// TIA Portal V16 export
// export: Created 2022-11-17T15:49:23.5959361Z, ExportSetting WithDefaults, DisplayName Totally Integrated Automation Portal, DisplayVersion V16 Update 6, DisplayName TIA Portal Version Control Interface, DisplayVersion V16 Update 2, DisplayName TIA Portal Openness, DisplayVersion V16 Update 6, DisplayName SINAMICS Startdrive Advanced, DisplayVersion V16 Update 5, DisplayName SINAMICS Startdrive G130, G150, S120, S150, SINAMICS MV, S210, DisplayVersion V16 Update 5, DisplayName SINAMICS Startdrive G110M, G120, G120C, G120D, G120P, G115D, DisplayVersion V16 Update 5, DisplayName STEP 7 Professional, DisplayVersion V16 Update 6, DisplayName STEP 7 Safety, DisplayVersion V16, DisplayName WinCC Advanced, DisplayVersion V16 Update 6
FUNCTION "FC34_SafetyBarrierStd" : Void   // FC34, LAD
{ S7_Optimized_Access := 'FALSE' }
VERSION : 0.1
// stored: AutoNumber false, IsIECCheckEnabled false, SetENOAutomatically false, UDAEnableTagReadback false
BEGIN

REGION Network 1: Alarm 24: Emergency on infeed safety barrier (Barrier)
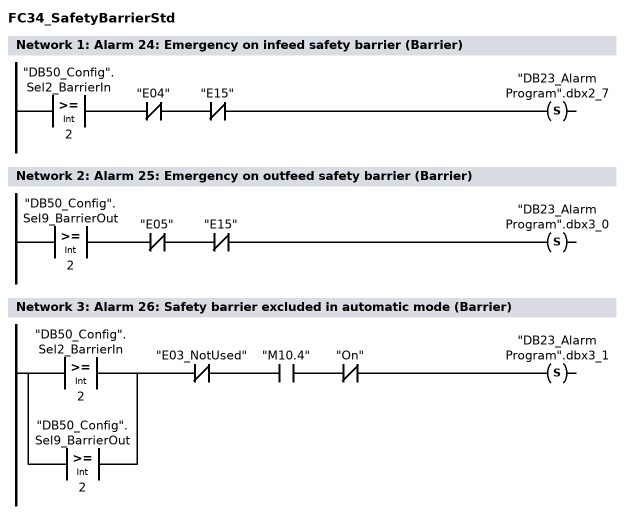
   RUNG wire#powerrail
      { S7_Templates := "SrcType := Int" } GE_Contact(in1 := "DB50_Config".Sel2_BarrierIn, in2 := 2)
      I_Contact( "E04" )
      I_Contact( "E15" )
      S_Coil( "DB23_AlarmProgram".dbx2_7 )
   END_RUNG
   // the same network as SCL:
   IF ("DB50_Config".Sel2_BarrierIn >= 2) AND NOT "E04" AND NOT "E15" THEN
       "DB23_AlarmProgram".dbx2_7 := TRUE;
   END_IF;
END_REGION

REGION Network 2: Alarm 25: Emergency on outfeed safety barrier (Barrier)
   RUNG wire#powerrail
      { S7_Templates := "SrcType := Int" } GE_Contact(in1 := "DB50_Config".Sel9_BarrierOut, in2 := 2)
      I_Contact( "E05" )
      I_Contact( "E15" )
      S_Coil( "DB23_AlarmProgram".dbx3_0 )
   END_RUNG
   // the same network as SCL:
   IF ("DB50_Config".Sel9_BarrierOut >= 2) AND NOT "E05" AND NOT "E15" THEN
       "DB23_AlarmProgram".dbx3_0 := TRUE;
   END_IF;
END_REGION

REGION Network 3: Alarm 26: Safety barrier excluded in automatic mode (Barrier)
   RUNG wire#powerrail
      { S7_Templates := "SrcType := Int" } GE_Contact(in1 := "DB50_Config".Sel2_BarrierIn, in2 := 2)
      wire#w1
      I_Contact( "E03_NotUsed" )
      Contact( "M10.4" )
      I_Contact( "On" )
      S_Coil( "DB23_AlarmProgram".dbx3_1 )
   END_RUNG
   RUNG wire#powerrail
      { S7_Templates := "SrcType := Int" } GE_Contact(in1 := "DB50_Config".Sel9_BarrierOut, in2 := 2)
   END_RUNG wire#w1
   // the same network as SCL:
   IF (("DB50_Config".Sel2_BarrierIn >= 2) OR ("DB50_Config".Sel9_BarrierOut >= 2)) AND NOT "E03_NotUsed" AND "M10.4" AND NOT "On" THEN
       "DB23_AlarmProgram".dbx3_1 := TRUE;
   END_IF;
END_REGION
END_FUNCTION
